// TIA Portal V19 export
TYPE "IPC_Msg_Send_Err"
   STRUCT
      TimeOut_ACK : Bool;   // Flag timeout comunicazione IPC - nessuna risposta entro PT_TIMEOUT
      BufferShift : Struct   // Gestione errori durante compattazione buffer con MOVE_BLK_VARIANT
         Error : Bool;   // TRUE = errore durante spostamento, buffer potenzialmente inconsistente
         ErrCode : Int;   // Codice errore specifico restituito da MOVE_BLK_VARIANT per diagnostica Gestione messaggi rifiutati dall'IPC (ACK negativo) con meccanismo retry
      END_STRUCT;
      Msg_NotAccepted : Struct   // Gestione messaggi rifiutati dall'IPC (ACK negativo) con meccanismo retry
         Presence : Bool;   // TRUE = messaggio in attesa di retry dopo rifiuto
         Code_ACK : DInt;   // Codice errore IPC (es: -1=malformato, -2=topic invalid, ecc.)
         Msg : "IPC_Msg_Generico";   // Copia del messaggio rifiutato per analisi e retry
      END_STRUCT;
   END_STRUCT;
END_TYPE
